FUNCTION_BLOCK PUBLIC FB_PizzaAmericanStyle IMPLEMENTS I_Pizza
VAR_INPUT
END_VAR
VAR_OUTPUT
END_VAR
VAR
END_VAR

METHOD GetDescription : STRING
GetDescription := 'Pizza American Style:';
END_METHOD

METHOD GetPrice : LREAL
GetPrice := 4.2;
END_METHOD

END_FUNCTION_BLOCK

(* stored: Version 1.1.0.1, ProductVersion 3.1.4022.16
   POU FB_PizzaAmericanStyle: Id {7d348bba-5d27-45fb-98e9-4b97ebd77ada}, SpecialFunc None
   Method GetDescription: Id {61d94432-215f-4c4e-93a5-37042a71622e}
   Method GetPrice: Id {0cca242f-c731-4f97-ae5c-d14bb340b421} *)
